// Mitsubishi GX Works2 project: automation_proj   PLC: FX3G

// global labels: Global1
VAR_GLOBAL
  master_on AT X007 : BOOL;
  system_break AT M0 : BOOL;
  working_status AT Y007 : BOOL;
  em_off AT X005 : BOOL;
  strawberry_stock AT D1100 : REAL;
  lemon_stock AT D1102 : REAL;
  stabilizer_stock AT D1104 : REAL;
END_VAR
VAR_GLOBAL CONSTANT
  strawberry_per_regular : REAL := 40.0;
  lemon_per_regular : REAL := 65.0;
  stabilizer_per_regular : REAL := 15.0;
  strawberry_per_extra : REAL := 55.0;
  lemon_per_extra : REAL := 95.0;
END_VAR
VAR_GLOBAL
  gummy_stock AT D1106 : REAL;
END_VAR
VAR_GLOBAL CONSTANT
  gummy_per_regular : REAL := 4.0;
  gummy_per_extra : REAL := 10.0;
  units_per_package : REAL := 7.0;
END_VAR
VAR_GLOBAL
  flavor_making_start AT X001 : BOOL;
  analog_type_picker AT D8280 : INT;
  strawberry_for_curr_batch AT D1108 : REAL;
  lemon_for_curr_batch AT D1110 : REAL;
  stabilizer_for_curr_batch AT D1112 : REAL;
  gummy_for_curr_batch AT D1114 : REAL;
  test AT Y011 : BOOL;
  is_extra AT M1 : BOOL;
END_VAR
VAR_GLOBAL CONSTANT
  stabilizer_per_extra : REAL := 30.0;
END_VAR
VAR_GLOBAL
  analog_read AT D8200 : INT;
  flavor_preperation AT Y000 : BOOL;
  preperation_break AT M2 : BOOL;
  preparing_timer_c AT TC0 : BOOL;
  preparing_timer_n AT TN0 : INT;
  preparing_timer_s AT TS0 : BOOL;
  start_cooling AT X002 : BOOL;
  cooling_indicator AT Y002 : BOOL;
  temp_sensor AT X003 : BOOL;
  cooling_timer_c AT TC1 : BOOL;
  cooling_timer_n AT TN1 : INT;
  cooling_timer_s AT TS1 : BOOL;
  initial_strawberry AT D1116 : REAL;
  initial_lemon AT D1118 : REAL;
  initial_stabilizer AT D1120 : REAL;
  initial_gummy AT D1122 : REAL;
  mixing_ready AT M3 : BOOL;
  mixing_time AT D1124 : REAL;
  mixing_timer_c AT TC2 : BOOL;
  mixing_timer_n AT TN2 : INT;
  mixing_timer_s AT TS2 : BOOL;
  mixing_lamp_a AT Y005 : BOOL;
  mixing_lamp_b AT Y006 : BOOL;
  alternating_lamps_helper AT M4 : BOOL;
  alt_lamp_timer_a_c AT TC3 : BOOL;
  alt_lamp_timer_a_n AT TN3 : INT;
  alt_lamp_timer_a_s AT TS3 : BOOL;
  alt_lamp_timer_b_c AT TC4 : BOOL;
  alt_lamp_timer_b_n AT TN4 : INT;
  alt_lamp_timer_b_s AT TS4 : BOOL;
  cooling_ready AT M5 : BOOL;
  total_packages AT D1126 : REAL;
  total_p_output AT D8282 : INT;
  mixing_indicator AT M6 : BOOL;
  strawberry_cooling_container AT D1128 : REAL;
  lemon_cooling_container AT D1130 : REAL;
  mixing_container AT D1132 : REAL;
END_VAR
VAR_GLOBAL CONSTANT
  regular_s_ic_weight : REAL := 50.0;
  regular_l_ic_weight : REAL := 70.0;
  extra_s_ic_weight : REAL := 80.0;
  extra_l_ic_weight : REAL := 100.0;
  single_gummy_weight : REAL := 7.0;
END_VAR

// task Task_01 (event TRUE, interval 0, priority 31): POU_01

PROGRAM POU_01
(* structured ladder/FBD written out as ST: instructions are called as NAME(EN, inputs, outputs); _pN, _eN, _tN stand for wires *)
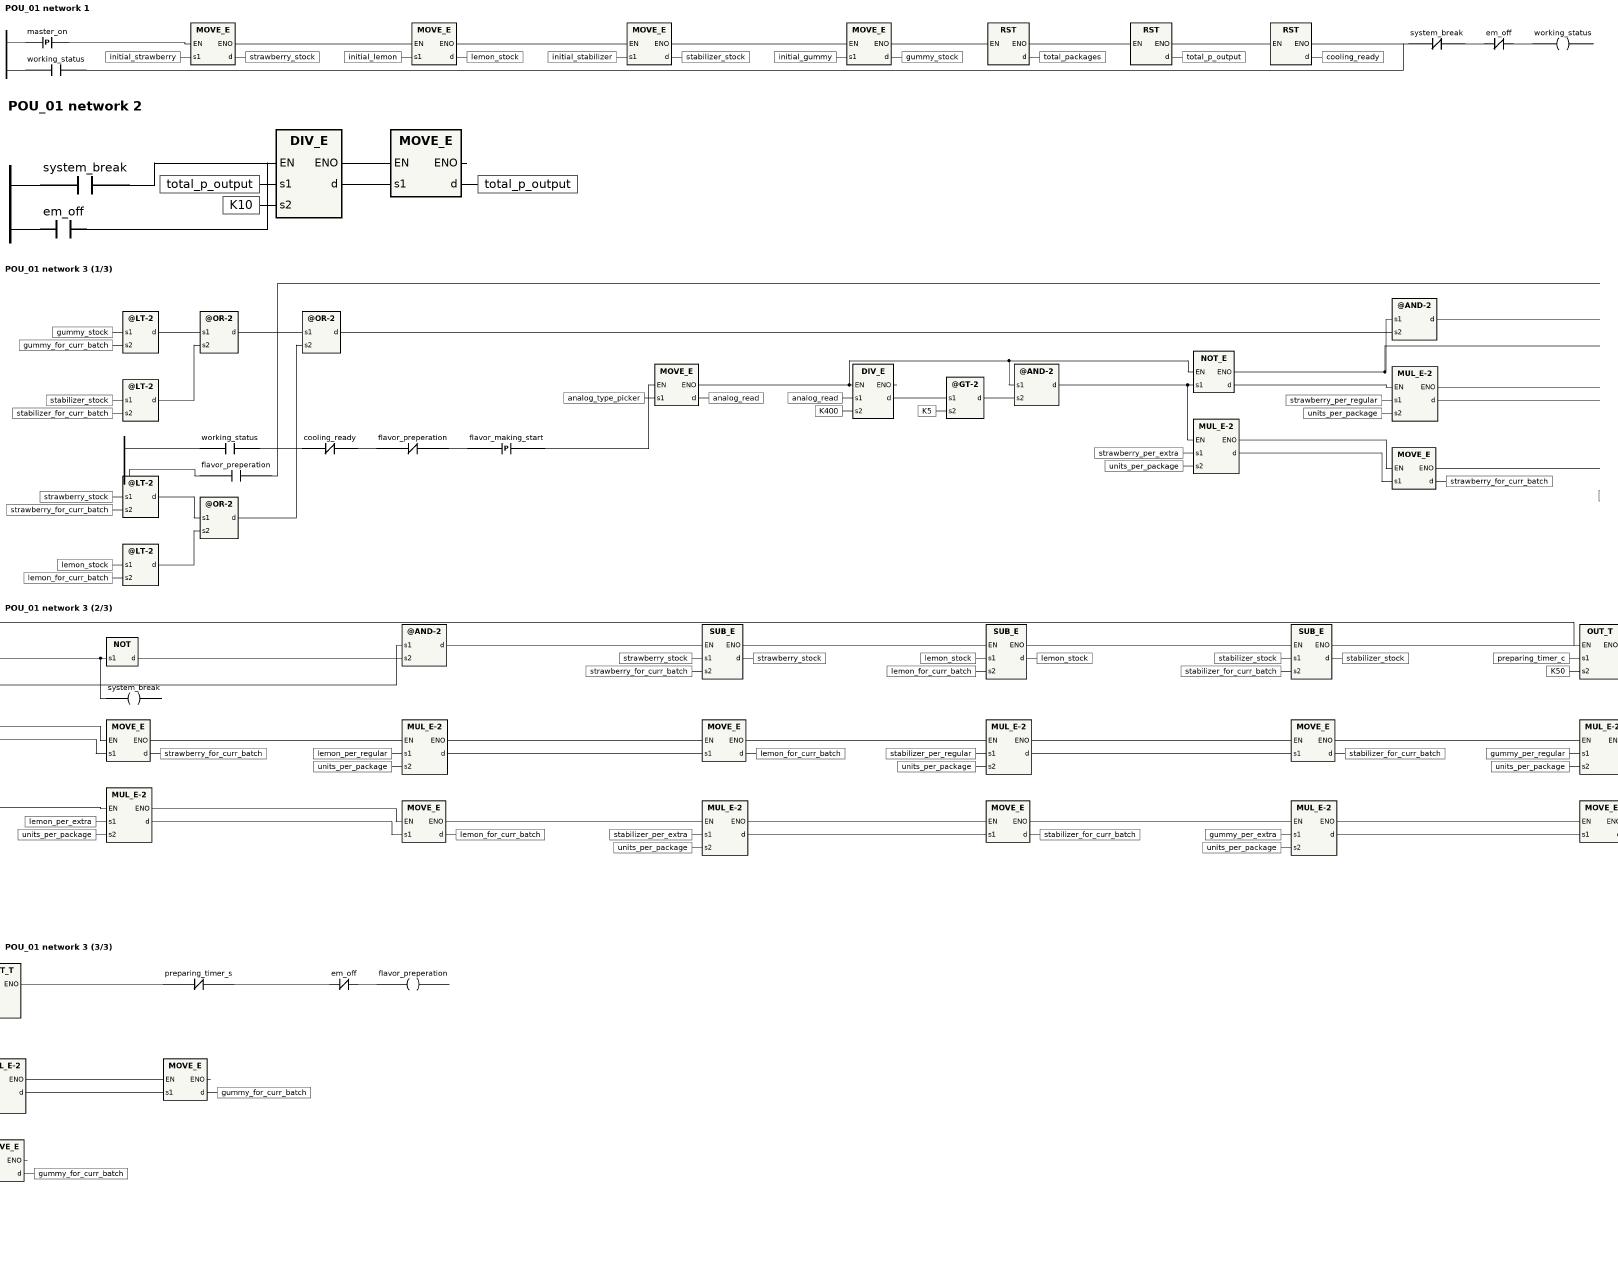
(* network 1 *)
_e1 := MOVE_E(LDP(TRUE, master_on), initial_strawberry, strawberry_stock);
_e2 := MOVE_E(_e1, initial_lemon, lemon_stock);
_e3 := MOVE_E(_e2, initial_stabilizer, stabilizer_stock);
_e4 := MOVE_E(_e3, initial_gummy, gummy_stock);
_e5 := RST(_e4, total_packages);
_e6 := RST(_e5, total_p_output);
_e7 := RST(_e6, cooling_ready);
working_status := ((_e7 OR working_status) AND NOT system_break) AND NOT em_off;
(* network 2 *)
_e2 := DIV_E(system_break OR em_off, total_p_output, K10, _t1);
MOVE_E(_e2, _t1, total_p_output);
(* network 3 *)
_e1 := MOVE_E(working_status AND NOT cooling_ready AND NOT flavor_preperation AND LDP(TRUE, flavor_making_start), analog_type_picker, analog_read);
DIV_E(_e1, analog_read, K400, _t2);
_p3 := @AND-2(_e1, @GT-2(_t2, K5));
_e5 := NOT_E(_e1, _p3, _t4);
_p6 := @AND-2(_e5, @OR-2(@OR-2(@LT-2(gummy_stock, gummy_for_curr_batch), @LT-2(stabilizer_stock, stabilizer_for_curr_batch)), @OR-2(@LT-2(strawberry_stock, strawberry_for_curr_batch), @LT-2(lemon_stock, lemon_for_curr_batch))));
_e7 := SUB_E(@AND-2(_e5, NOT(_p6)), strawberry_stock, strawberry_for_curr_batch, strawberry_stock);
_e8 := SUB_E(_e7, lemon_stock, lemon_for_curr_batch, lemon_stock);
_e9 := SUB_E(_e8, stabilizer_stock, stabilizer_for_curr_batch, stabilizer_stock);
_e10 := OUT_T(_e9 OR flavor_preperation, preparing_timer_c, K50);
flavor_preperation := _e10 AND NOT preparing_timer_s AND NOT em_off;
_e12 := MUL_E(_t4, strawberry_per_regular, units_per_package, _t11);
_e13 := MOVE_E(_e12, _t11, strawberry_for_curr_batch);
_e15 := MUL_E(_e13, lemon_per_regular, units_per_package, _t14);
_e16 := MOVE_E(_e15, _t14, lemon_for_curr_batch);
_e18 := MUL_E(_e16, stabilizer_per_regular, units_per_package, _t17);
_e19 := MOVE_E(_e18, _t17, stabilizer_for_curr_batch);
_e21 := MUL_E(_e19, gummy_per_regular, units_per_package, _t20);
MOVE_E(_e21, _t20, gummy_for_curr_batch);
_e23 := MUL_E(_p3, strawberry_per_extra, units_per_package, _t22);
_e24 := MOVE_E(_e23, _t22, strawberry_for_curr_batch);
_e26 := MUL_E(_e24, lemon_per_extra, units_per_package, _t25);
_e27 := MOVE_E(_e26, _t25, lemon_for_curr_batch);
_e29 := MUL_E(_e27, stabilizer_per_extra, units_per_package, _t28);
_e30 := MOVE_E(_e29, _t28, stabilizer_for_curr_batch);
system_break := _p6;
_e32 := MUL_E(_e30, gummy_per_extra, units_per_package, _t31);
MOVE_E(_e32, _t31, gummy_for_curr_batch);
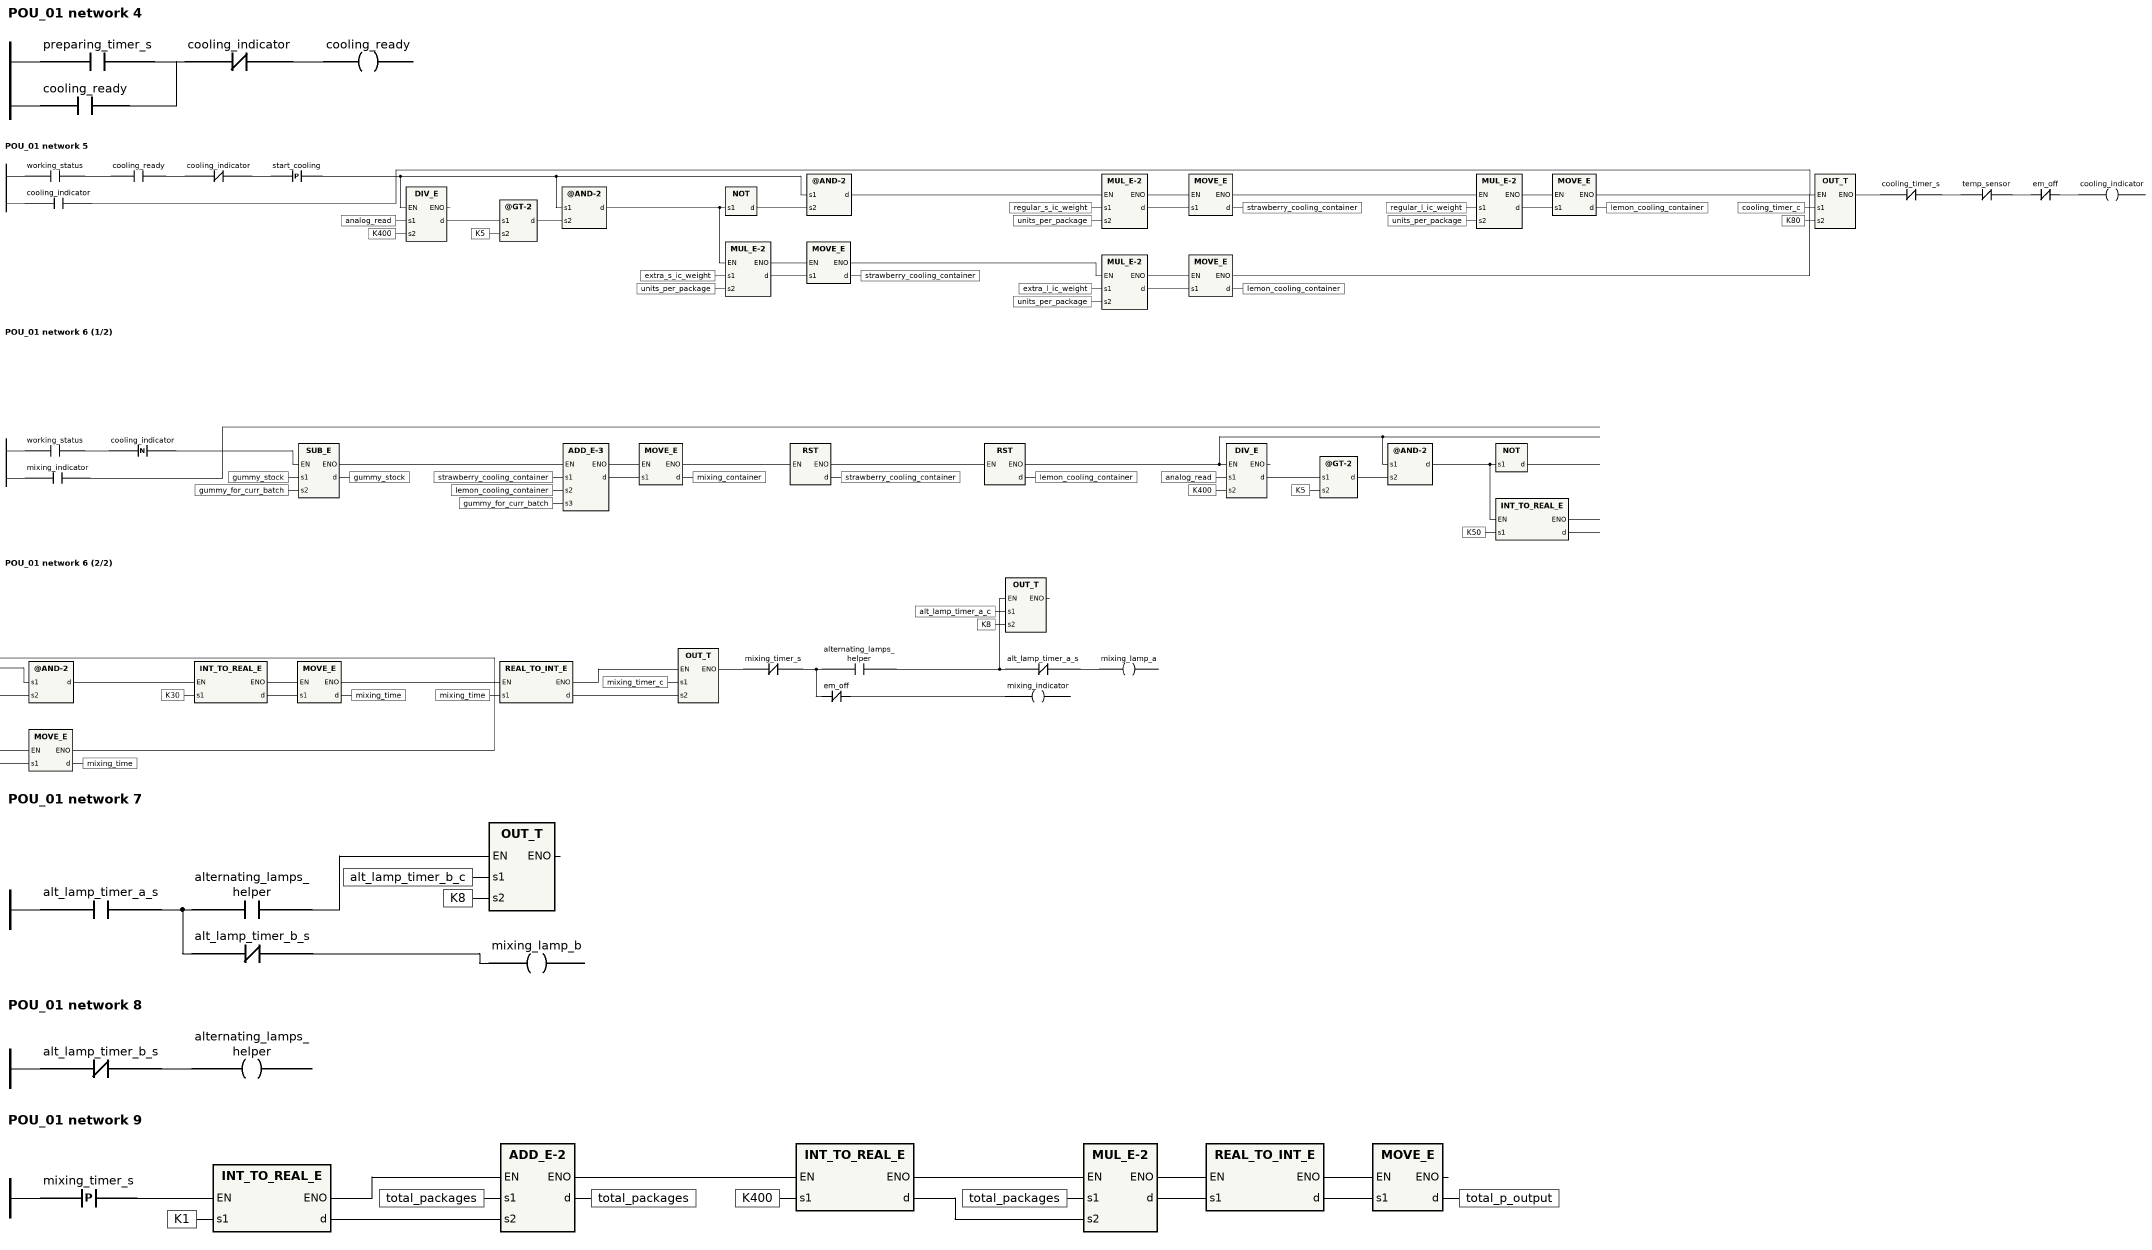
(* network 4 *)
cooling_ready := (preparing_timer_s OR cooling_ready) AND NOT cooling_indicator;
(* network 5 *)
_p1 := working_status AND cooling_ready AND NOT cooling_indicator AND LDP(TRUE, start_cooling);
DIV_E(_p1, analog_read, K400, _t2);
_p3 := @AND-2(_p1, @GT-2(_t2, K5));
_e5 := MUL_E(@AND-2(_p1, NOT(_p3)), regular_s_ic_weight, units_per_package, _t4);
_e6 := MOVE_E(_e5, _t4, strawberry_cooling_container);
_e8 := MUL_E(_e6, regular_l_ic_weight, units_per_package, _t7);
_e9 := MOVE_E(_e8, _t7, lemon_cooling_container);
_e11 := MUL_E(_p3, extra_s_ic_weight, units_per_package, _t10);
_e12 := MOVE_E(_e11, _t10, strawberry_cooling_container);
_e14 := MUL_E(_e12, extra_l_ic_weight, units_per_package, _t13);
_e15 := MOVE_E(_e14, _t13, lemon_cooling_container);
_e16 := OUT_T(_e9 OR _e15 OR cooling_indicator, cooling_timer_c, K80);
cooling_indicator := _e16 AND NOT cooling_timer_s AND NOT temp_sensor AND NOT em_off;
(* network 6 *)
_e1 := SUB_E(working_status AND LDF(TRUE, cooling_indicator), gummy_stock, gummy_for_curr_batch, gummy_stock);
_e3 := ADD_E(_e1, strawberry_cooling_container, lemon_cooling_container, gummy_for_curr_batch, _t2);
_e4 := MOVE_E(_e3, _t2, mixing_container);
_e5 := RST(_e4, strawberry_cooling_container);
_e6 := RST(_e5, lemon_cooling_container);
DIV_E(_e6, analog_read, K400, _t7);
_p8 := @AND-2(_e6, @GT-2(_t7, K5));
_e10 := INT_TO_REAL_E(@AND-2(_e6, NOT(_p8)), K30, _t9);
_e11 := MOVE_E(_e10, _t9, mixing_time);
_e13 := INT_TO_REAL_E(_p8, K50, _t12);
_e14 := MOVE_E(_e13, _t12, mixing_time);
_e16 := REAL_TO_INT_E(_e11 OR _e14 OR mixing_indicator, mixing_time, _t15);
_e17 := OUT_T(_e16, mixing_timer_c, _t15);
_p18 := _e17 AND NOT mixing_timer_s;
_p19 := _p18 AND alternating_lamps_helper;
OUT_T(_p19, alt_lamp_timer_a_c, K8);
mixing_lamp_a := _p19 AND NOT alt_lamp_timer_a_s;
mixing_indicator := _p18 AND NOT em_off;
(* network 7 *)
OUT_T(alt_lamp_timer_a_s AND alternating_lamps_helper, alt_lamp_timer_b_c, K8);
mixing_lamp_b := alt_lamp_timer_a_s AND NOT alt_lamp_timer_b_s;
(* network 8 *)
alternating_lamps_helper := NOT alt_lamp_timer_b_s;
(* network 9 *)
_e2 := INT_TO_REAL_E(LDP(TRUE, mixing_timer_s), K1, _t1);
_e3 := ADD_E(_e2, total_packages, _t1, total_packages);
_e5 := INT_TO_REAL_E(_e3, K400, _t4);
_e7 := MUL_E(_e5, total_packages, _t4, _t6);
_e9 := REAL_TO_INT_E(_e7, _t6, _t8);
MOVE_E(_e9, _t8, total_p_output);
END_PROGRAM
